FUNCTION_BLOCK FB_PitchSoftLimits
VAR_INPUT
	Pitch	:	HOMS_PitchMechanismOld;
END_VAR
VAR_OUTPUT
	xHiLS	:	BOOL;
	xLoLS	:	BOOL;
END_VAR
VAR
	diHys	:	DINT := 500; //500 nm (1 inc/nm)
	STO: BOOL;
END_VAR

STO := Pitch.Stepper.diInputs.3;

xHiLS S= Pitch.diEncCnt < Pitch.diEncPosLimHi - diHys;
xHiLS R= Pitch.diEncCnt > Pitch.diEncPosLimHi;

xLoLS S= Pitch.diEncCnt > Pitch.diEncPosLimLo + diHys;
xLoLS R= Pitch.diEncCnt < Pitch.diEncPosLimLo;

xHiLS := xHiLS AND STO;
xLoLS := xLoLS AND STO;

END_FUNCTION_BLOCK

(* stored: Version 1.1.0.1, ProductVersion 3.1.4022.18
   POU FB_PitchSoftLimits: Id {3b9899a1-d7a0-44d6-9210-b3d8d5950ecd}, SpecialFunc None *)
